Staubli VAL3: onBackSpace.pgx

program onBackSpace(tool& x_tTool[])
begin
  //
  // NB sEvent is the selected
  // element in the LIST
  //
  if nIndex==0
    call editTool(x_tTool)
    call tcp:setTool(x_tTool,nIndexTool)
    logMsg("[KERNEL] INTERFACE:Change value of the tool :"+toString("",nIndexTool))
  endIf
  //
end
